ABB RobotStudio station: version1.rsstn

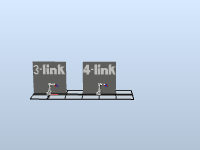
Station version1 (saved by RobotStudio format 3)
Controller System
  mechanical unit ROB_1: IRB120_3_58__01, 6 joints, base frame (0, 0, 0) mm
  mechanical unit ROB_2: IRB120_3_58__01_2, 6 joints, base frame (3000, 0, 0) mm
Layout (positions relative to the parent item):
  - IRB120_3_58__01 [mechanism, from Robots\IRB120_3_58_G_01.rslib] at (0, 0, 0) mm; joint values [0, 0, 0, 0, 0.5236, 0] (rad or m)
  - IRB120_3_58__01_2 [mechanism, from Robots\IRB120_3_58_G_01.rslib] at (3000, 0, 0) mm; joint values [0, 0, 0, 0, 0.5236, 0] (rad or m)
  - MyNewTool [mechanism, from Libraries\Tool_1rslib.rslib] at (364.35, 0, 594) mm, rotated rx 180 ry 60 rz 180 deg
  - MyNewTool_2 [mechanism, from Libraries\Tool_1rslib.rslib] at (3364.35, 0, 594) mm, rotated rx 180 ry 60 rz 180 deg
  - Wall [part, from Libraries\Wall.rslib] at (-1000, 150, 0) mm
  - Wall2 [part, from Libraries\Wall2.rslib] at (0, 150, 0) mm
  - 3 [part, from Libraries\3.rslib] at (-203.1, 0, 2640.47) mm, rotated rx 90 ry 0 rz 0 deg
  - 4 [part, from Libraries\4.rslib] at (2237.05, 0, 3057.64) mm, rotated rx 90 ry 0 rz 0 deg
  - hyphen [part, from Libraries\hifen.rslib] at (2501.1, 0, 1530.78) mm, rotated rx 90 ry 0 rz 0 deg
  - hyphen_2 [part, from Libraries\hifen.rslib] at (-579.72, 0, 1530.78) mm, rotated rx 90 ry 0 rz 0 deg
  - i [part, from Libraries\i.rslib] at (6.71, 0, 2650.44) mm, rotated rx 90 ry 0 rz 0 deg
  - i_2 [part, from Libraries\i.rslib] at (3065.42, 0, 2650.44) mm, rotated rx 90 ry 0 rz 0 deg
  - k [part, from Libraries\k.rslib] at (0, 0, 2646.78) mm, rotated rx 90 ry 0 rz 0 deg
  - k_2 [part, from Libraries\k.rslib] at (3032.61, 0, 2646.78) mm, rotated rx 90 ry 0 rz 0 deg
  - l [part, from Libraries\l.rslib] at (-369.34, 0, 1257.2) mm, rotated rx 90 ry 0 rz 0 deg
  - l_2 [part, from Libraries\l.rslib] at (2704.62, 0, 1257.2) mm, rotated rx 90 ry 0 rz 0 deg
  - n [part, from Libraries\n.rslib] at (0, 0, 2647.94) mm, rotated rx 90 ry 0 rz 0 deg
  - n_2 [part, from Libraries\n.rslib] at (3053.54, 0, 2647.94) mm, rotated rx 90 ry 0 rz 0 deg
Attachment: MyNewTool is attached to IRB120_3_58__01 / Link6
Attachment: MyNewTool_2 is attached to IRB120_3_58__01_2 / Link6
Targets, tools, work objects and paths stored in the station, written as RAPID:
! task T_ROB1
MODULE CalibData
  PERS tooldata Tool_1:=[TRUE,[[0,150,105],[1,0,0,0]],[1,[0,0,1],[1,0,0,0],0,0,0]];
ENDMODULE

! task T_ROB1
MODULE Action
  VAR jointtarget joints:=[[0,0,0,0,0,0],[9E9,9E9,9E9,9E9,9E9,9E9]];
  PROC ReadingArm()
  ENDPROC
  PROC ReadingAng()
  ENDPROC
  PROC pWriteSomething()
  ENDPROC
  PROC WI()
  ENDPROC
  PROC main()
    ReadingArm;
    ReadingAng;
    WI;
    MoveAbsJ joints,v1000,fine,Tool_1\WObj:=wobj0;
    pWriteSomething;
  ENDPROC
ENDMODULE

! task T_ROB2
MODULE CalibData
  PERS tooldata Tool_1:=[TRUE,[[0,150,105],[1,0,0,0]],[1,[0,0,1],[1,0,0,0],0,0,0]];
ENDMODULE

! task T_ROB2
MODULE Action2
  VAR jointtarget joints:=[[0,0,0,0,0,0],[9E9,9E9,9E9,9E9,9E9,9E9]];
  PROC ReadingArm()
  ENDPROC
  PROC ReadingAng()
  ENDPROC
  PROC pWriteSomething()
  ENDPROC
  PROC WI()
  ENDPROC
  PROC main()
    ReadingArm;
    ReadingAng;
    WI;
    MoveAbsJ joints,v1000,fine,Tool_1\WObj:=wobj0;
    pWriteSomething;
  ENDPROC
ENDMODULE

